{attribute 'qualified_only'}
{attribute 'strict'}
{attribute 'to_string'}
TYPE MotionDirection :
(
    Positive,
    ShortestWay,
    Negative,
    Current,
    Undefined
);
END_TYPE

(* stored: Version 1.1.0.1
   DUT MotionDirection: Id {bfa94b18-f414-4de2-8278-f984d418aba9} *)
